PROGRAM PRG_SAF
VAR
END_VAR

Nc2MasterAxis();

END_PROGRAM

(* stored: Version 1.1.0.1
   POU PRG_SAF: Id {6efa3269-2dd8-426c-804d-06e18b3a07f0}, SpecialFunc None *)
